// TIA Portal project "ENSAYO FC MOV-B" (V11)

(* hardware
DEVICE "S7300/ET200 station_1"  SIMATIC 300-Station
   slot 0: "Perfil soporte_0"  Rail  6ES7 390-1***0-0AA0
   slot 2: "PLC_1"  CPU 313C-2 DP  6ES7 313-6CF03-0AB0  V2.6
      slot 0: "Interfaz MPI_1"  MPI
      slot 1: "Interfaz DP_1"  DP
      slot 2: "DI16/DO16_1"  DI16/DO16
      slot 4: "Contaje_1"  Counter
*)

// ===== PLC "PLC_1"  CPU 313C-2 DP =====

VAR_GLOBAL   // PLC tag table "Tabla de variables estándar"
   "Tag_1" AT %I0.0 : Bool;
   "Tag_2" AT %I0.1 : Bool;
   "Tag_3" AT %I0.2 : Bool;
   "Tag_4" AT %I0.3 : Bool;
   "Tag_5" AT %Q0.0 : Bool;
   "Tag_6" AT %Q0.1 : Bool;
   "Tag_7" AT %Q0.2 : Bool;
   "Tag_8" AT %Q0.3 : Bool;
   "Tag_9" AT %MB0 : Byte;
   "Tag_10" AT %M0.0 : Bool;
   "Tag_11" AT %M0.1 : Bool;
   "Tag_12" AT %M0.2 : Bool;
   "Tag_13" AT %M0.3 : Bool;
END_VAR

DATA_BLOCK "DATOS"   // DB1
{ S7_Optimized_Access := 'FALSE' }
VERSION : 0.1
   VAR
      CONTROL : Byte;
      FLANCOS : Array [0..7] of Bool;
   END_VAR
BEGIN
END_DATA_BLOCK

FUNCTION "M0V-B" : Void   // FC1, LAD
{ S7_Optimized_Access := 'FALSE' }
VERSION : 0.1
   VAR_INPUT
      "1" : Bool;
      "2" : Bool;
      "3" : Bool;
      "4" : Bool;
   END_VAR
   VAR_OUTPUT
      "A" : Byte;
   END_VAR
   VAR_TEMP   // added for the SCL form of the ladder/FBD networks
      _w1 : Bool;
   END_VAR
BEGIN

REGION Network 1
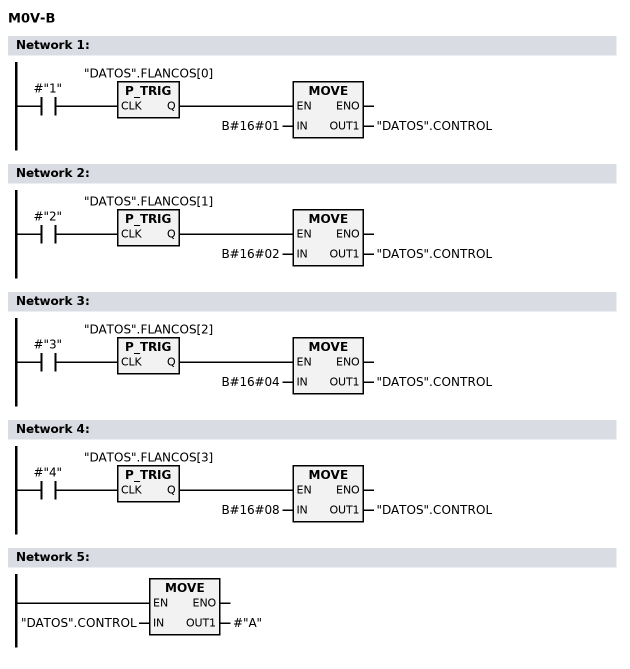
   RUNG wire#powerrail
      Contact( #"1" )
      P_Trig( "DATOS".FLANCOS[0] )
      { S7_GenerateENO := "TRUE" } Move(in := B#16#01, out1 => "DATOS".CONTROL)
   END_RUNG
   // the same network as SCL:
   #_w1 := #"1" AND NOT "DATOS".FLANCOS[0];   // rising edge
   "DATOS".FLANCOS[0] := #"1";
   IF #_w1 THEN "DATOS".CONTROL := B#16#01; END_IF;
END_REGION

REGION Network 2
   RUNG wire#powerrail
      Contact( #"2" )
      P_Trig( "DATOS".FLANCOS[1] )
      { S7_GenerateENO := "TRUE" } Move(in := B#16#02, out1 => "DATOS".CONTROL)
   END_RUNG
   // the same network as SCL:
   #_w1 := #"2" AND NOT "DATOS".FLANCOS[1];   // rising edge
   "DATOS".FLANCOS[1] := #"2";
   IF #_w1 THEN "DATOS".CONTROL := B#16#02; END_IF;
END_REGION

REGION Network 3
   RUNG wire#powerrail
      Contact( #"3" )
      P_Trig( "DATOS".FLANCOS[2] )
      { S7_GenerateENO := "TRUE" } Move(in := B#16#04, out1 => "DATOS".CONTROL)
   END_RUNG
   // the same network as SCL:
   #_w1 := #"3" AND NOT "DATOS".FLANCOS[2];   // rising edge
   "DATOS".FLANCOS[2] := #"3";
   IF #_w1 THEN "DATOS".CONTROL := B#16#04; END_IF;
END_REGION

REGION Network 4
   RUNG wire#powerrail
      Contact( #"4" )
      P_Trig( "DATOS".FLANCOS[3] )
      { S7_GenerateENO := "TRUE" } Move(in := B#16#08, out1 => "DATOS".CONTROL)
   END_RUNG
   // the same network as SCL:
   #_w1 := #"4" AND NOT "DATOS".FLANCOS[3];   // rising edge
   "DATOS".FLANCOS[3] := #"4";
   IF #_w1 THEN "DATOS".CONTROL := B#16#08; END_IF;
END_REGION

REGION Network 5
   RUNG wire#powerrail
      { S7_GenerateENO := "TRUE" } Move(in := "DATOS".CONTROL, out1 => #"A")
   END_RUNG
   // the same network as SCL:
   #"A" := "DATOS".CONTROL;
END_REGION
END_FUNCTION

ORGANIZATION_BLOCK "Main"   // OB1, LAD
TITLE = "Main Program Sweep (Cycle)"
{ S7_Optimized_Access := 'FALSE' }
VERSION : 0.1
   VAR_TEMP
      OB1_EV_CLASS : Byte;   // Bits 0-3 = 1 (Coming event), Bits 4-7 = 1 (Event class 1)
      OB1_SCAN_1 : Byte;   // 1 (Cold restart scan 1 of OB 1), 3 (Scan 2-n of OB 1)
      OB1_PRIORITY : Byte;   // Priority of OB Execution
      OB1_OB_NUMBR : Byte;   // 1 (Organization block 1, OB1)
      OB1_RESERVED_1 : Byte;   // Reserved for system
      OB1_RESERVED_2 : Byte;   // Reserved for system
      OB1_PREV_CYCLE : Int;   // Cycle time of previous OB1 scan (milliseconds)
      OB1_MIN_CYCLE : Int;   // Minimum cycle time of OB1 (milliseconds)
      OB1_MAX_CYCLE : Int;   // Maximum cycle time of OB1 (milliseconds)
      OB1_DATE_TIME : Date_And_Time;   // Date and time OB1 started
   END_VAR
BEGIN

REGION Network 1
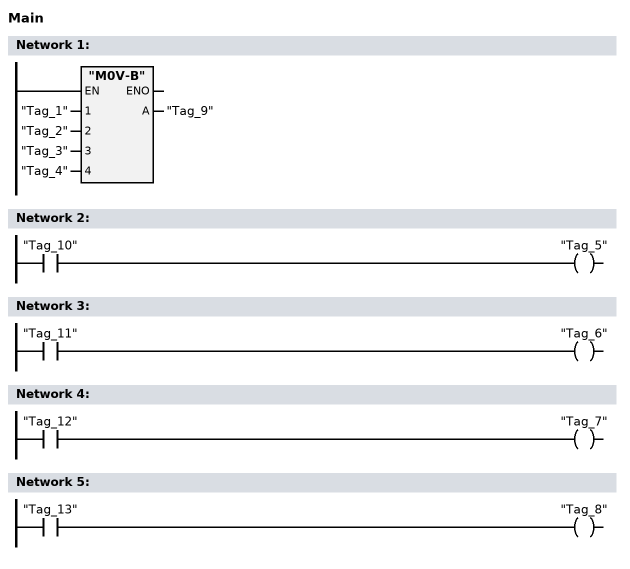
   RUNG wire#powerrail
      "M0V-B"("1" := "Tag_1", "2" := "Tag_2", "3" := "Tag_3", "4" := "Tag_4", "A" => "Tag_9")
   END_RUNG
   // the same network as SCL:
   "M0V-B"("1" := "Tag_1", "2" := "Tag_2", "3" := "Tag_3", "4" := "Tag_4", "A" => "Tag_9");
END_REGION

REGION Network 2
   RUNG wire#powerrail
      Contact( "Tag_10" )
      Coil( "Tag_5" )
   END_RUNG
   // the same network as SCL:
   "Tag_5" := "Tag_10";
END_REGION

REGION Network 3
   RUNG wire#powerrail
      Contact( "Tag_11" )
      Coil( "Tag_6" )
   END_RUNG
   // the same network as SCL:
   "Tag_6" := "Tag_11";
END_REGION

REGION Network 4
   RUNG wire#powerrail
      Contact( "Tag_12" )
      Coil( "Tag_7" )
   END_RUNG
   // the same network as SCL:
   "Tag_7" := "Tag_12";
END_REGION

REGION Network 5
   RUNG wire#powerrail
      Contact( "Tag_13" )
      Coil( "Tag_8" )
   END_RUNG
   // the same network as SCL:
   "Tag_8" := "Tag_13";
END_REGION
END_ORGANIZATION_BLOCK